Universal Robots PolyScope program: move_path_2.urp

Program move_path_2 (installation=default directory=/programs createdIn=5.14.5 lastSavedIn=5.14.5 robotSerialNumber=20236801216)
Calibrated DH parameters: a=[-0.000021, -0.748897, -0.28186, -0.00004, -0.000055, 0]; d=[0.236225, -424.082933, -1564.66872, 1988.95162, 0.159094, 0.153873]; alpha=[1.570844, 0.001002, 0.000337, 1.571488, -1.569996, 0]; deltaTheta=[0, -0.516316, 5.626292, 1.173211, 0.000001, 0]
InitVariablesNode
Robot Program (runOnlyOnce=false)
  pa1 := path1[1]
  pa2 := path1[2]
  p1 := path1[3]
  p2 := path1[4]
  p3 := path1[5]
  p4 := path1[6]
  p5 := path1[7]
  pr1 := path1[8]
  pvr1 := path1[12]
  pvr2 := path1[13]
  MoveJ speed 60 deg/s, acceleration 80 deg/s^2 (useActiveTCP=true) feature=Base
    SuppressedNode
      Waypoint Waypoint_9: TCP in base x=-308.524 y=606.099 z=242.383 mm, rx=-0.1348 ry=-3.0618 rz=-0.0522 rad; joints [-82.604, -97.742, 135.138, 229.977, -86.039, -167.57] deg; TCP offset x=0 y=0 z=260 mm, rx=0 ry=0 rz=0 rad
    Waypoint Waypoint_7: TCP in base x=-308.522 y=606.103 z=242.387 mm, rx=1.3699 ry=1.0669 rz=-1.2572 rad; joints [-84.673, -56.548, 94.558, 52.545, 94.971, 14.541] deg; TCP offset x=8.55 y=-265.17 z=108.77 mm, rx=1.2092 ry=-1.2092 rz=1.2092 rad
  MoveJ speed 60 deg/s, acceleration 80 deg/s^2 (useActiveTCP=true) feature=Base
    Waypoint Variable (Variable): variable=pa1
  MoveL speed 200 mm/s, acceleration 1200 mm/s^2 (useActiveTCP=true) feature=Base
    Waypoint Variable (Variable): variable=pa2
  MoveL speed 50 mm/s, acceleration 1200 mm/s^2 (useActiveTCP=true) feature=Base
    Waypoint Variable (Variable): variable=p1
  Wait Sleep waitTime=1
  MoveL speed 12 mm/s, acceleration 1200 mm/s^2 (useActiveTCP=true) feature=Base
    Waypoint Variable (Variable): variable=p2
  MoveP speed 0.5 mm/s, acceleration 500 mm/s^2 (blendRadius=0.001 useActiveTCP=true) feature=Base
    CircleMove (OrientationMode=FIXED)
      Waypoint Variable (Variable): variable=p3
      Waypoint Variable (Variable): variable=p4
  MoveL speed 12 mm/s, acceleration 1200 mm/s^2 (useActiveTCP=true) feature=Base
    Waypoint Variable (Variable): variable=p5
  MoveL speed 250 mm/s, acceleration 1200 mm/s^2 (useActiveTCP=true) feature=Base
    Waypoint Variable (Variable): variable=pr1
  SuppressedNode
    MoveJ speed 60 deg/s, acceleration 80 deg/s^2 (useActiveTCP=true) feature=Base
      Waypoint Waypoint_8: TCP in base x=-372.861 y=716.17 z=314.677 mm, rx=1.5708 ry=0 rz=0 rad; joints [-79.161, -60.426, 105.047, -44.564, -79.226, 359.93] deg; TCP offset x=0 y=0 z=19 mm, rx=0 ry=0 rz=0 rad
  MoveL speed 250 mm/s, acceleration 1200 mm/s^2 (useActiveTCP=true) feature=Base
    Waypoint Variable (Variable): variable=pvr1
